(* IEC 61131-3 sources: ics/BLR1_PhoenixContact/BLR1_AXC1050_21/LogicalPOUs/MISC, 5 files *)

(* ---- PlsFlwCnt.ST ---- *)
(*@PROPERTIES_EX@
TYPE: POU
LOCALE: 0
IEC_LANGUAGE: ST
PLC_TYPE: independent
PROC_TYPE: independent
GROUP: MISC.FB
*)
(*@KEY@:DESCRIPTION*)

(*@KEY@:END_DESCRIPTION*)
FUNCTION_BLOCK PlsFlwCnt

(*Group:Default*)

VAR
	Tick :	BOOL;
	TickCount :	INT;
	TicksNum :	REAL;
	CounterPulse :	R_TRIG;
END_VAR

VAR_INPUT
	Pls :	BOOL;
	PulseWeight :	REAL;
END_VAR

VAR_OUTPUT
	Flow :	REAL;
END_VAR

(*@KEY@: WORKSHEET
NAME: PlsFlwCnt
IEC_LANGUAGE: ST
*)
Tick:= not Tick;

IF Tick THEN
	TickCount:= TickCount + 1;
	Tick:= false;
END_IF;

IF TickCount > 6000 THEN
	TickCount:= 0;
	TicksNum:= 0.0;
	Flow:= 0.0;
END_IF;

CounterPulse(CLK:= Pls);

IF CounterPulse.Q THEN
	TicksNum:= int_to_real(TickCount);
	TickCount:= 0;
	Flow:= (PulseWeight * 360000.0) / (TicksNum + 1.0);
END_IF;

(*@KEY@: END_WORKSHEET *)
END_FUNCTION_BLOCK

(* ---- GAS_CNT.ST ---- *)
(*@PROPERTIES_EX@
TYPE: POU
LOCALE: 0
IEC_LANGUAGE: ST
PLC_TYPE: independent
PROC_TYPE: independent
GROUP: MISC
*)
(*@KEY@:DESCRIPTION*)

(*@KEY@:END_DESCRIPTION*)
PROGRAM GAS_CNT

(*Group:Default*)

VAR_EXTERNAL
	AI :	SENSOR;
END_VAR

VAR
	Blr1GasCntFB :	PlsFlwCnt;
	Blr2GasCntFB :	PlsFlwCnt;
	Blr3GasCntFB :	PlsFlwCnt;
END_VAR

VAR_EXTERNAL
	Blr11_GasFlowPls :	BOOL;
	Blr12_GasFlowPls :	BOOL;
	Blr13_GasFlowPls :	BOOL;
END_VAR

(*@KEY@: WORKSHEET
NAME: GAS_CNT
IEC_LANGUAGE: ST
*)
Blr1GasCntFB(Pls:=Blr11_GasFlowPls,PulseWeight:=1.0);
AI[116].Ymax:= Blr1GasCntFB.Flow * 1.4;

Blr2GasCntFB(Pls:=Blr12_GasFlowPls,PulseWeight:=1.0);
AI[117].Ymax:= Blr2GasCntFB.Flow * 1.4;

Blr3GasCntFB(Pls:=Blr13_GasFlowPls,PulseWeight:=1.0);
AI[118].Ymax:= Blr3GasCntFB.Flow * 1.4;

(*@KEY@: END_WORKSHEET *)
END_PROGRAM

(* ---- TICK_100MS.ST ---- *)
(*@PROPERTIES_EX@
TYPE: POU
LOCALE: 0
IEC_LANGUAGE: ST
PLC_TYPE: independent
PROC_TYPE: independent
GROUP: MISC
*)
(*@KEY@:DESCRIPTION*)

(*@KEY@:END_DESCRIPTION*)
PROGRAM TICK_100MS

(*Group:Default*)

VAR
	RS_1 :	RS;
	R_TRIG_1 :	R_TRIG;
END_VAR

VAR_EXTERNAL
	TICK_100MS :	BOOL;
	TICK_100MS_PLS :	BOOL;
END_VAR

(*@KEY@: WORKSHEET
NAME: TICK_100MS
IEC_LANGUAGE: ST
*)
RS_1(SET:= not TICK_100MS,RESET1:=TICK_100MS);
TICK_100MS:=RS_1.Q1;

R_TRIG_1(CLK:=TICK_100MS);
TICK_100MS_PLS:=R_TRIG_1.Q;

(*@KEY@: END_WORKSHEET *)
END_PROGRAM

(* ---- TICK_1S.ST ---- *)
(*@PROPERTIES_EX@
TYPE: POU
LOCALE: 0
IEC_LANGUAGE: ST
PLC_TYPE: independent
PROC_TYPE: independent
GROUP: MISC
*)
(*@KEY@:DESCRIPTION*)

(*@KEY@:END_DESCRIPTION*)
PROGRAM TICK_1S

(*Group:Default*)

VAR
	RS_1 :	RS;
END_VAR

VAR_EXTERNAL
	TICK_1S :	BOOL;
END_VAR

VAR
	R_TRIG_1 :	R_TRIG;
END_VAR

VAR_EXTERNAL
	TICK_1S_PLS :	BOOL;
END_VAR

(*@KEY@: WORKSHEET
NAME: TICK_1S
IEC_LANGUAGE: ST
*)
RS_1(SET:= not TICK_1S,RESET1:= TICK_1S);
TICK_1S:=RS_1.Q1;

R_TRIG_1(CLK:= TICK_1S);
TICK_1S_PLS:=R_TRIG_1.Q;

(*@KEY@: END_WORKSHEET *)
END_PROGRAM

(* ---- TimeTicks.ST ---- *)
(*@PROPERTIES_EX@
TYPE: POU
LOCALE: 0
IEC_LANGUAGE: ST
PLC_TYPE: independent
PROC_TYPE: independent
GROUP: MISC
*)
(*@KEY@:DESCRIPTION*)

(*@KEY@:END_DESCRIPTION*)
PROGRAM TimeTicks

(*Group:Default*)

VAR
	ton100MS :	TON;
	pls100MS :	R_TRIG;
	ton1S :	TON;
	pls1S :	R_TRIG;
END_VAR

VAR_EXTERNAL
	TICK_100MS :	BOOL;
	TICK_1S :	BOOL;
END_VAR

(*@KEY@: WORKSHEET
NAME: TimeTicks
IEC_LANGUAGE: ST
*)

(*================================================================================================*)
(*100ms tick*)
(*================================================================================================*)
ton100MS(IN:= not ton100MS.Q ,PT:= t#100ms);
pls100MS(CLK:= ton100MS.Q);
TICK_100MS:= pls100MS.Q;

(*================================================================================================*)
(*1s tick*)
(*================================================================================================*)
ton1S(IN:=not ton1S.Q,PT:= t#1s);
pls1S(CLK:= ton1S.Q);
TICK_1S:=pls1S.Q;

(*@KEY@: END_WORKSHEET *)
END_PROGRAM
